VAR_GLOBAL
END_VAR

(* stored: Version 1.1.0.1, ProductVersion 3.1.4018.5
   GVL GVL: Id {4b504377-0bb2-4e94-b82c-1948a3ff8f19} *)
